FUNCTION F_TemperatureMonitorSetpoints : ST_TemperatureMonitorSetpoints
VAR_INPUT
END_VAR
VAR
	stTempMonSP : ST_TemperatureMonitorSetpoints := (fMaxTemperature := 40);
END_VAR

F_TemperatureMonitorSetpoints := stTempMonSP;

END_FUNCTION

(* stored: Version 1.1.0.1, ProductVersion 3.1.4020.14
   POU F_TemperatureMonitorSetpoints: Id {29bceff7-0180-4c10-ba9c-150191a55fd0}, SpecialFunc None *)
